
TYPE "Axis3D_001"
STRUCT
        X : "MotorStatus_001";
        Y : "MotorStatus_001";
        Z : "MotorStatus_001";
        POSITION : ARRAY[0..2] OF REAL;
        VELOCITY : ARRAY[0..2] OF REAL;
END_STRUCT;
END_TYPE